FUNCTION F_Homing : BOOL
VAR
	LoopCount	: INT := 2000;
END_VAR

END_FUNCTION

(* stored: Version 1.1.0.1, ProductVersion 3.1.4024.11
   POU F_Homing: Id {306e44f6-bc33-4124-bfd9-c6ad82f7dfc7}, SpecialFunc None *)
